RoboDK station: station.rdk

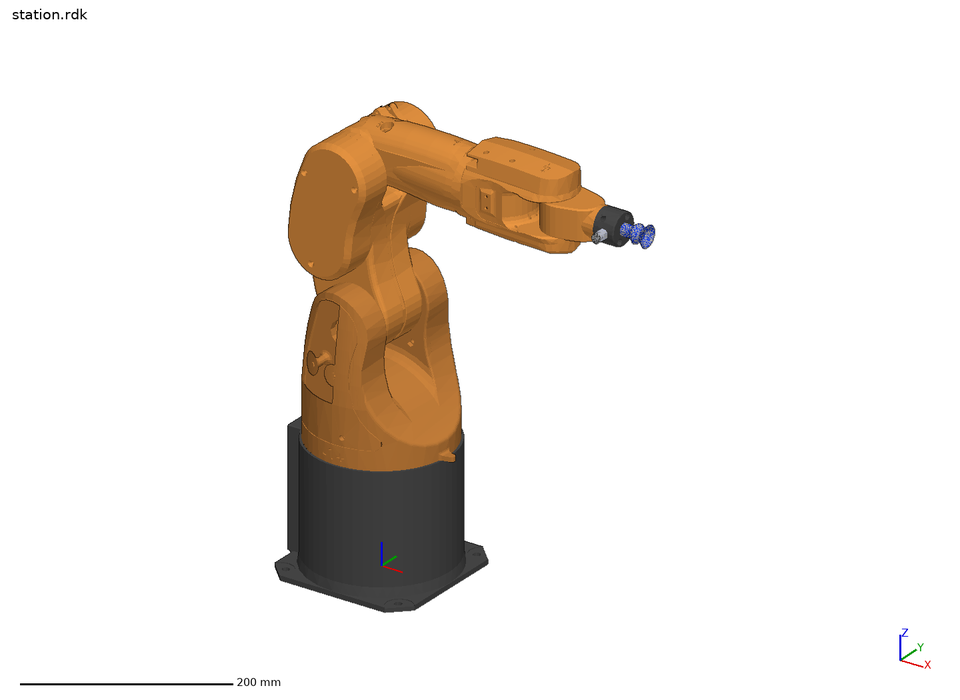
[picture v0: the station drawn from its stored meshes, robots at their saved joint values, targets as dots, program paths as lines]
Station station (saved by RoboDK 5.2.4). Poses are relative to the parent item; angles as X-Y-Z fixed-axis rotations.
  - frame K1.1 Osiris Base at (0, 0, 0) mm
    - robot K1.1 Osiris: 6 axes
        modified DH rows (alpha deg, a mm, theta deg, d mm): 0, 0, 0, 256.25; -90, -11.87, -90, 0; 0, 175, 0, 0; -90, 3.98, 0, 216; 90, 0, 0, 0; -90, 0, 0, 63
        joint limits [-175, -90, -180, -200, -90, -2000] to [175, 120, 30, 200, 90, 2000]; home [0, 0, 0, 0, 0, 0]; saved at [-3.037, 0.094, -0.094, 89.999, -3.037, -89.999]
      - tool Suction head, TCP at (0, 0, 50) mm, size 35 x 49 x 45.3 mm
